{attribute 'linkalways'} 
{attribute 'no_explicit_call' := 'This FB is a CLASS and must be accessed using methods or properties'}
{attribute 'enable_dynamic_creation'}
FUNCTION_BLOCK FINAL MOD_USINT EXTENDS Node
VAR
	in1 : _USINT(0);
	in2 : _USINT(0);
	out : _USINT(0);
END_VAR

METHOD PUBLIC Clone : I_Node
VAR
	pNode : POINTER TO MOD_USINT;
END_VAR
pNode := __NEW(MOD_USINT);
Clone := pNode^;
END_METHOD

METHOD FB_init : BOOL
VAR_INPUT
	bInitRetains : BOOL; // if TRUE, the retain variables are initialized (warm start / cold start)
	bInCopyCode : BOOL;  // if TRUE, the instance afterwards gets moved into the copy code (online change)
END_VAR
AddInput('in1',THIS^.in1);
AddInput('in2',THIS^.in2);
AddOutput('out', THIS^.out);
END_METHOD

METHOD PROTECTED OnExecute
VAR
END_VAR
out.Value := in1.Value MOD in2.Value;
END_METHOD

END_FUNCTION_BLOCK

(* stored: Version 1.1.0.1, ProductVersion 3.1.4024.15
   POU MOD_USINT: Id {b6aff697-dfc1-4a66-b436-2a66871a5cc0}, SpecialFunc None
   Folder Constructor: Id {fa613f73-278a-497c-841a-2523fac16f5d}
   Method Clone: Id {0c3213d9-3cb6-4b34-a51b-6445d0fe31ce}
   Method FB_init: Id {74f3708e-2159-4a92-a116-c32273cebd7d}
   Method OnExecute: Id {03cca6bb-34fd-42b8-987a-f6f03f007610} *)
